// TIA Portal V17 export
// export: Created 2024-08-09T12:53:18.5899957Z, ExportSetting WithDefaults, DisplayName Totally Integrated Automation Portal, DisplayVersion V17 Update 7, DisplayName TIA Portal Openness, DisplayVersion V17 Update 7, DisplayName TIA Portal Version Control Interface, DisplayVersion V17, DisplayName STEP 7 Professional, DisplayVersion V17 Update 7, DisplayName STEP 7 Safety, DisplayVersion V17 Update 6, DisplayName WinCC Professional, DisplayVersion V17 Update 7
TYPE "S_Cir_Trans"
// stored: IsFailsafeCompliant false
   STRUCT
      Pt_Zs : "S_Suivi_Dosage";
      DosCommun { S7_SetPoint := 'True'} : "S_Dosage_Commun";
      Circuit { S7_SetPoint := 'True'} : "S_Circuit";
      Dial_Def : "S_DIALOG_DEF";
      Lst_Att_Aval_Libre { S7_SetPoint := 'True'} : Array[0.."T_MAX_AMONTAVAL"] of "S_TacheNiv";
      Lst_Att_Auto_Demar { S7_SetPoint := 'True'} : Array[0.."T_MAX_AMONTAVAL"] of "S_TacheNiv";
      Lst_Att_Fin_Amont { S7_SetPoint := 'True'} : Array[0.."T_MAX_AMONTAVAL"] of "S_TacheNiv";
      Lst_Taches_Amont_Qte { S7_SetPoint := 'True'} : Array[0.."T_MAX_AMONTAVAL"] of SInt;
      Num_Circuit { S7_SetPoint := 'True'} : USInt;
      Origine : USInt;
      Destination : USInt;
   END_STRUCT;
   // Lst_Taches_Amont_Qte[0..9] := -1;
END_TYPE
